{attribute 'qualified_only'}
VAR_GLOBAL
DoorClosed : BOOL; (*Is true when door is closed*)
TapOpen : BOOL; (*Is true when tap is open*)
DesiredTemperature : BOOL; (*Is true when water is at desired temperature*)
ShowerON : BOOL; (*Is true when shower is running*)
StartTimer : TIME; (*Starts a timer when shower is running*)
StopTimer : TIME; (*Stops shower when timer expires*)
CurrentTime : TIME; (*Displays current time left to shower*)
MaxShowerTime : TIME := T#0.25M; (*Maximum time allowed to shower*)
END_VAR

(* stored: Version 1.1.0.1, ProductVersion 3.1.4024.12
   GVL GVL: Id {4cad470e-3bd1-47d6-ab6d-168c6f1adafd} *)
